FUNCTION_BLOCK FB_SimpleTcpTaskQueue
VAR_INPUT
END_VAR
VAR_OUTPUT
END_VAR
VAR
	WaitingQueue		: FB_MemRingBufferEx;
	ArrWaitingQueue		: ARRAY[0..MAXBUFFERSIZE] OF ST_TcpTaskBuffer;
	ActingQueue			: FB_MemRingBufferEx;
	ArrActingQueue		: ARRAY[0..MAXBUFFERSIZE] OF ST_TcpTaskBuffer;
	
	PushTask	: ST_TcpTask;
	PopTask		: ST_TcpTask;
	EmptyTask	: ST_TcpTask;
	
	StepTaskConsume : DINT;
	
	_NoTaskToConsume : BOOL;
	_WaitingForTaskDone: BOOL;
	
	_TaskComplete : BOOL;
	
	_WaitingTaskCount: UDINT;
	_WaitingUsedSize: UDINT;
	_WaitingFreeSize: UDINT;
	
	_ActingTaskCount: UDINT;
	_ActingTotalSize: UDINT;
	_ActingFreeSize: UDINT;

END_VAR

VAR CONSTANT
	MAXBUFFERSIZE: UDINT := 128;
END_VAR

WaitingQueue(pWrite:= , cbWrite:= , pBuffer:= ADR(ArrWaitingQueue), cbBuffer:= SIZEOF(ArrWaitingQueue), 
	bOk=> , pRead=> , cbRead=> , nCount=> _WaitingTaskCount, cbSize=> _WaitingUsedSize, cbFree=> _WaitingFreeSize);
ActingQueue(pWrite:= , cbWrite:= , pBuffer:= ADR(ArrActingQueue), cbBuffer:= SIZEOF(ArrActingQueue), 
	bOk=> , pRead=> , cbRead=> , nCount=> _ActingTaskCount, cbSize=> _ActingTotalSize, cbFree=> _ActingFreeSize);

_NoTaskToConsume := (StepTaskConsume = 0);
_WaitingForTaskDone := (StepTaskConsume <> 0);
CASE StepTaskConsume OF
	0:
	_NoTaskToConsume := TRUE;
	IF ActingQueue.nCount <> 0 THEN
		StepTaskConsume := 10;
	END_IF
	
	10:
	ActingQueue.A_GetHead(pWrite:= , cbWrite:= , pBuffer:= ADR(ArrActingQueue), cbBuffer:= SIZEOF(ArrActingQueue), 
	bOk=> , pRead=> , cbRead=> , nCount=> _ActingTaskCount, cbSize=> _ActingTotalSize, cbFree=> _ActingFreeSize);
	IF ActingQueue.bOk THEN
		MEMCPY(destAddr:= ADR(PopTask), srcAddr:= ActingQueue.pRead, n:= MIN(SIZEOF(PopTask),ActingQueue.cbRead));
		_TaskComplete := FALSE;
		StepTaskConsume := 20;
	ELSE
		StepTaskConsume := 0;
	END_IF
	
	20:
	// wait for task done
	
END_CASE

PROPERTY ActingTaskCount : UDINT
GET
ActingTaskCount := _ActingTaskCount;
END_GET
END_PROPERTY

METHOD AddActingTask : BOOL
VAR_INPUT
	TaskName : STRING(24);
	TaskType : INT; (* 0:Once, 1:Regular *)
	TaskData : ARRAY[0..255] OF BYTE;
END_VAR
PushTask.TaskName := TaskName;
PushTask.TaskType := TaskType;
PushTask.TaskData := TaskData;
ActingQueue.A_AddTail(pWrite:= ADR(PushTask), cbWrite:= SIZEOF(PushTask), pBuffer:= ADR(ArrActingQueue), cbBuffer:= SIZEOF(ArrActingQueue), 
	bOk=> AddActingTask, pRead=> , cbRead=> , nCount=> _ActingTaskCount, cbSize=> _ActingTotalSize, cbFree=> _ActingFreeSize);
END_METHOD

PROPERTY CurrentTask : ST_TcpTask
GET
CurrentTask := PopTask;
END_GET
END_PROPERTY

METHOD FinishTask : BOOL
VAR_INPUT
END_VAR
ActingQueue.A_FreeHead(pWrite:= , cbWrite:= , pBuffer:= ADR(ArrActingQueue), cbBuffer:= SIZEOF(ArrActingQueue), 
bOk=> , pRead=> , cbRead=> , nCount=> _ActingTaskCount, cbSize=> _ActingTotalSize, cbFree=> _ActingFreeSize);
IF ActingQueue.bOk THEN
	MEMCPY(destAddr:= ADR(PopTask), srcAddr:= ADR(EmptyTask), n:= SIZEOF(ST_TcpTask));
	IF ActingQueue.nCount <> 0 THEN
		StepTaskConsume := 10;
	ELSE
		StepTaskConsume := 0;
	END_IF
END_IF
END_METHOD

END_FUNCTION_BLOCK

(* stored: Version 1.1.0.1, ProductVersion 3.1.4024.12
   POU FB_SimpleTcpTaskQueue: Id {a0d5a2a5-6bce-4f1c-8f88-35110661d4b1}, SpecialFunc None
   Property ActingTaskCount: Id {2d194400-93bb-48de-a175-4c53fba06ee5}
   Get Get: Id {35890d36-03e8-453f-8325-e7fa9fcbf85e}
   Method AddActingTask: Id {1a5b38e8-3e79-49e3-a824-2bb22cd5c11d}
   Property CurrentTask: Id {ea68b0af-5181-4df7-baa5-140dba78ddd8}
   Get Get: Id {21624ead-e38d-4bc5-81b5-bf6f65f8d593}
   Method FinishTask: Id {e9707e9b-7715-4f8b-897f-ce08e6ac7c5e} *)
